FUNCTION_BLOCK FB_RobotMovementTime
VAR_INPUT
	inm_Couting				:BOOL;
	inint_FirstStation		:INT	:=-1;
	inint_SecondStation		:INT	:=-1;
END_VAR
VAR_OUTPUT
	outs_MovementTime		:TYPE_MovementTime;
END_VAR
VAR
	rt_TimeActive			:R_TRIG;
	ft_TimeActive			:F_TRIG;
	t_StartTime				:TIME;
	
END_VAR

rt_TimeActive(CLK:=inm_Couting);

IF rt_TimeActive.Q
	THEN
	t_StartTime:=TIME();
END_IF

ft_TimeActive(CLK:=inm_Couting);

IF ft_TimeActive.Q
	THEN
	outs_MovementTime.FirstStation:=inint_FirstStation;
	outs_MovementTime.SecondStation:=inint_SecondStation;
	outs_MovementTime.MovementTime:=TIME_TO_REAL(TIME() - t_StartTime)/1000;
END_IF

END_FUNCTION_BLOCK

(* stored: Version 1.1.0.1, ProductVersion 3.1.4024.3
   POU FB_RobotMovementTime: Id {f1249df3-61aa-4489-8b11-cfaeec635c41}, SpecialFunc None *)
